Yaskawa INFORM job: R1-S1-SAMPLE.JBI

/JOB
//NAME R1-S1-SAMPLE
//POS
///NPOS 5,0,5,0,0,0
///TOOL 0
///POSTYPE PULSE
///PULSE
C00000=0,-22155,-18106,0,-17887,0
C00001=-6348,-38367,-29889,-13986,-20076,6564
C00002=-5697,-22758,-19385,-13694,-18452,6429
C00003=-5697,-22758,-19385,-13694,-18452,6429
C00004=-5697,-22758,-19385,-13694,-18452,6429
EC00000=-29914,247808
EC00001=-29914,247808
EC00002=-29914,247808
EC00003=-14293,247808
EC00004=-14293,247808
//INST
///DATE 2023/01/18 18:12
///ATTR SC,RW
///GROUP1 RB1
///GROUP2 ST1
NOP
MOVJ C00000 VJ=0.78  +MOVJ EC00000 VJ=0.78
MOVJ C00001 VJ=0.78  +MOVJ EC00001 VJ=0.78
MOVL C00002 V=11.0  +MOVJ EC00002 VJ=0.78
SMOVL C00003 V=11.0  +MOVJ EC00003
MOVJ C00004 VJ=0.78  +MOVJ EC00004 VJ=0.78
END
